{attribute 'qualified_only'}
{attribute 'strict'}
TYPE E_NCI_CHANNEL_ERROR :
(
  e_Null,
  e_InvalidReference_ChannelRef,
  e_AxisConfigurationMismatch_McAxis,
  e_AxisConfigurationMismatch_AuxAxis


);
END_TYPE

(* stored: Version 1.1.0.1
   DUT E_NCI_CHANNEL_ERROR: Id {1122f668-1b0d-4766-af41-16a534c31d15} *)
